PROGRAM SequencyControl
VAR
	index:WORD;
END_VAR

CASE SEQ.iSeqStepN OF 
	 0:    //INIT
		 SEQ.sSeqStepDescription:='Init';
		 SEQ.bSeqStep_TaskDone[0]:=VAL.bAllValves_At_Home AND Cell.bHousingPresent AND Cell.bPalmButton;  //trigger the sequency
		 IF SEQ.bSeqStepN_TaskDone_DelayDone[0] THEN
			 FOR index:=1 TO SEQ.iStepN DO
				 SEQ.bSeqStep_TaskDone[index]:=FALSE;
			 END_FOR
			 seq.iSeqStepN:=5;
		 END_IF
	5:
		 SEQ.sSeqStepDescription:='Loading parts to hoursing';
		 SEQ.bSeqStep_TaskDone[5]:=VAL.bValve_A_AtWorkSensor;
		 IF SEQ.bSeqStepN_TaskDone_DelayDone[5] THEN
			 FOR index:=6 TO SEQ.iStepN DO
				 SEQ.bSeqStep_TaskDone[index]:=FALSE;
			 END_FOR
			 seq.iSeqStepN:=10;
		 END_IF
	10:
		 SEQ.sSeqStepDescription:='Clamp house';
		 SEQ.bSeqStep_TaskDone[10]:=VAL.bValve_A_AtWorkSensor AND VAl.bValve_B_AtWorkSensor;
		 IF SEQ.bSeqStepN_TaskDone_DelayDone[10] THEN
			 FOR index:=11 TO SEQ.iStepN DO
				 SEQ.bSeqStep_TaskDone[index]:=FALSE;
			 END_FOR
			 seq.iSeqStepN:=15;
		 END_IF
	15:
  	     SEQ.sSeqStepDescription:='Press/crimp the housing';
		 SEQ.bSeqStep_TaskDone[15]:=VAL.bValve_B_AtWorkSensor AND VAL.bValve_C_AtWorkSensor AND VAL.bValve_A_AtHomeSensor;
		 IF SEQ.bSeqStepN_TaskDone_DelayDone[15] THEN
			 FOR index:=0 TO SEQ.iStepN DO
				 SEQ.bSeqStep_TaskDone[index]:=FALSE;
			 END_FOR
			 seq.iSeqStepN:=20;
		 END_IF
	20:
  	     SEQ.sSeqStepDescription:='Open clamp';
		 SEQ.bSeqStep_TaskDone[20]:=VAl.bValve_B_AtHomeSensor;
		 IF SEQ.bSeqStepN_TaskDone_DelayDone[20] THEN
			 FOR index:=21 TO SEQ.iStepN DO
				 SEQ.bSeqStep_TaskDone[index]:=FALSE;
			 END_FOR
			 seq.iSeqStepN:=25;
		 END_IF
	25:  //work on cyl D
		 SEQ.sSeqStepDescription:='Heat houring for 10s';
		 SEQ.bSeqStep_TaskDone[25]:=VAL.bValve_D_AtWorkSensor AND VAL.bValve_C_AtWorkSensor;
		 IF SEQ.bSeqStepN_TaskDone_DelayDone[25] THEN
			 FOR index:=26 TO SEQ.iStepN DO
				 SEQ.bSeqStep_TaskDone[index]:=FALSE;
			 END_FOR
			 seq.iSeqStepN:=30;
		 END_IF
	30:  //home, home cyn C and Cyn B
		 SEQ.sSeqStepDescription:='Stop heat, open clamp';
		 SEQ.bSeqStep_TaskDone[30]:=VAL.bValve_C_AtHomeSensor AND VAL.bValve_D_AtHomeSensor;
		 IF SEQ.bSeqStepN_TaskDone_DelayDone[30] THEN
//			 FOR index:=26 TO SEQ.iStepN DO
//				 SEQ.bSeqStep_TaskDone[index]:=FALSE;
//			 END_FOR
			 seq.iSeqStepN:=0;
		 END_IF
END_CASE
SequencyCondition();

METHOD PUBLIC SequencyCondition : BOOL
VAR_INPUT
END_VAR
SEQ.fbSeqStepN_TaskDone_DelayTmr[0](IN:= SEQ.bSeqStep_TaskDone[0], PT:=T#2S , Q=>SEQ.bSeqStepN_TaskDone_DelayDone[0] );
SEQ.fbSeqStepN_TaskDone_DelayTmr[5](IN:= SEQ.bSeqStep_TaskDone[5], PT:=T#2S , Q=>SEQ.bSeqStepN_TaskDone_DelayDone[5] );
SEQ.fbSeqStepN_TaskDone_DelayTmr[10](IN:= SEQ.bSeqStep_TaskDone[10], PT:=T#2S , Q=>SEQ.bSeqStepN_TaskDone_DelayDone[10] );
SEQ.fbSeqStepN_TaskDone_DelayTmr[15](IN:= SEQ.bSeqStep_TaskDone[15], PT:=T#2S , Q=>SEQ.bSeqStepN_TaskDone_DelayDone[15] );
SEQ.fbSeqStepN_TaskDone_DelayTmr[20](IN:= SEQ.bSeqStep_TaskDone[20], PT:=T#2S , Q=>SEQ.bSeqStepN_TaskDone_DelayDone[20] );
SEQ.fbSeqStepN_TaskDone_DelayTmr[25](IN:= SEQ.bSeqStep_TaskDone[25], PT:=T#10S , Q=>SEQ.bSeqStepN_TaskDone_DelayDone[25] );
SEQ.fbSeqStepN_TaskDone_DelayTmr[30](IN:= SEQ.bSeqStep_TaskDone[30], PT:=T#2S , Q=>SEQ.bSeqStepN_TaskDone_DelayDone[30] );
END_METHOD

END_PROGRAM

(* stored: Version 1.1.0.1, ProductVersion 3.1.4024.12
   POU SequencyControl: Id {7dbeb3d8-e35b-4761-9a31-09968c80dca7}, SpecialFunc None
   Method SequencyCondition: Id {e73106a6-1c9e-4dba-ba76-41c8a3223427} *)
